Staubli VAL3: onExit.pgx

program onExit(bool& x_bSave[])
  local string l_sMessage
  local bool l_bYes
  local bool l_bCancel
  local string l_sButton[2]
begin

end
